// TIA Portal V17 export
// export: Created 2021-12-03T08:08:03.102286Z, ExportSetting WithDefaults, DisplayName Totally Integrated Automation Portal, DisplayVersion V17, DisplayName TIA Portal Openness, DisplayVersion V17, DisplayName TIA Portal Version Control Interface, DisplayVersion V17, DisplayName STEP 7 Professional, DisplayVersion V17, DisplayName STEP 7 Safety, DisplayVersion V17, DisplayName WinCC Advanced, DisplayVersion V17
VAR_GLOBAL   // PLC tag table "FailSafe_DI"
   "I_/EmStpAccCon_Ch1" AT %I40.0 : Bool;   // Emergency Stop Accelerator Console (True=No EmStp) / Консоль ускорителя канал 1
   "I_/EmStpP1_Ch1" AT %I40.1 : Bool;   // Emergency Stop Panel 1 (True=No EmStp) / Пульт Р1 канал 1
   "I_/EmStpP2_Ch1" AT %I40.2 : Bool;   // Emergency Stop Panel 2 (True=No EmStp) / Пульт Р2 канал 1
   I_PrDoor1Cls_Ch1 AT %I40.3 : Bool;   // Protecting Door 1 close / Замок блокирующий дверь 1 канал 1
   I_PrDoor2Cls_Ch1 AT %I40.4 : Bool;   // Protecting Door 2 close / Замок блокирующий дверь 2 канал 1
   "I_/EmStpDosimeter_Ch1" AT %I40.6 : Bool;   // Emergency Stop Dosimeter (True=No EmStp) / Дозиметр канал 1
   I_PrDoor1Req AT %I40.7 : Bool;   // Request Open Protecting Door 1 / Запрос на открытие двери 1
   I_P3AckInSArea_Ch1 AT %I41.0 : Bool;   // Panel 3: Acknowledgement in the Safety Area / Сброс внутри периметра безопасности
   I_FBPowerModulator AT %I41.1 : Bool;   // Feedback Contactor Modulator NA2-1Q3 / Обратная связь модулятора
   I_FBPowerConveyor AT %I41.2 : Bool;   // Feedback Contactor Freq. Converter Conveyor NA2-1Q7 / Обратная связь частотного преобразователя
   I_FBPowerXRayUnit AT %I41.3 : Bool;   // Feedback Contactor X-Ray Unit NA2-2Q7 / Обратная связь ускоритель
   I_PrDoor2Req AT %I42.3 : Bool;   // Request Open Protecting Door 2 / Запрос на открытие двери 2
   I_P1AckEmStpOutSArea AT %I42.4 : Bool;   // Panel 1: Acknowledgement Emergency Stop outsite the Safety Area / Сброс снаружи периметра безопасности
   I_FBPowerChiller AT %I42.5 : Bool;   // Feedback Contactor Chiller NA2-1Q5 / Обратная связь чиллер
   I_FBPower_AccConsol AT %I42.6 : Bool;   // Feedback Contactor Accelerator Console NA2-2Q3 / Обратная связь консоль ускорителя
   I_FBPowerModulator1P AT %I42.7 : Bool;   // Feedback Contactor Modulator 230VAC / Обратная связь модулятора 1 фаза
   "I_/EmStpP3_Ch1" AT %I60.0 : Bool;   // Emergency Stop Panel 3 (True=No EmStp) / Пульт P3 канал 1
   I_P2AgreeBut_Ch1 AT %I60.1 : Bool;   // Panel 2: Agree Button (True=Agree) / Кнопка разрешения канал 1
   I_P1KeyGenRel_Ch1 AT %I61.0 : Bool;   // Panel 1: Keyswitch General Release (True=Release) / Главный ключ разрешения канал 1
   I_P1KeyAccRel_Ch1 AT %I61.1 : Bool;   // Panel 1: Keyswitch Accelerator Release (Power Release Mod., X-Ray Unit, Acc.) / Ключ разрешения включения ускорителя канал 1
   I_Spare40_5 AT %I40.5 : Bool;   // Spare
   "I_/EmStpAccCon_Ch2" AT %I41.4 : Bool;   // Консоль ускорителя канал 2
   "I_/EmStpP1_Ch2" AT %I41.5 : Bool;   // Пульт Р1 канал 2
   "I_/EmStpP2_Ch2" AT %I41.6 : Bool;   // Пульт Р2 канал 2
   I_PrDoor1Cls_Ch2 AT %I41.7 : Bool;   // Замок блокирующий дверь 1 канал 2
   I_PrDoor2Cls_Ch2 AT %I42.0 : Bool;   // Замок блокирующий дверь 2 канал 2
   I_Spare42_1 AT %I42.1 : Bool;   // Spare
   I_Spare60_2 AT %I60.2 : Bool;   // Spare
   I_Spare60_3 AT %I60.3 : Bool;   // Spare
   I_Spare60_4 AT %I60.4 : Bool;   // Spare
   I_Spare60_5 AT %I60.5 : Bool;   // Spare
   I_Spare60_6 AT %I60.6 : Bool;   // Spare
   I_Spare60_7 AT %I60.7 : Bool;   // Spare
   I_Spare61_2 AT %I61.2 : Bool;   // Spare
   I_Spare61_3 AT %I61.3 : Bool;   // Spare
   "I_/EmStpP3_Ch2" AT %I61.4 : Bool;   // Пульт P3 канал 2
   I_P2AgreeBut_Ch2 AT %I61.5 : Bool;   // Кнопка разрешения канал 2
   I_Spare61_6 AT %I61.6 : Bool;   // Spare
   I_Spare61_7 AT %I61.7 : Bool;   // Spare
   "I_/EmStpDosimeter_Ch2" AT %I42.2 : Bool;   // Дозиметр канал 2
   I_Spare62_0 AT %I62.0 : Bool;   // Spare
   I_Spare62_1 AT %I62.1 : Bool;   // Spare
   I_Spare62_2 AT %I62.2 : Bool;   // Spare
   I_Spare62_3 AT %I62.3 : Bool;   // Spare
   I_P1KeyGenRel_Ch2 AT %I62.4 : Bool;   // Главный ключ разрешения канал 2
   I_P1KeyAccRel_Ch2 AT %I62.5 : Bool;   // Ключ разрешения включения ускорителя канал 2
   I_Spare62_6 AT %I62.6 : Bool;   // Spare
   I_Spare62_7 AT %I62.7 : Bool;   // Spare
END_VAR
